(* IEC 61131-3 sources: Industry-PLC-LLM/data/PLCBEAD_repo/PLCBEAD_PLCEmbed-main/PLC-BEAD/Source/GEB/Network_TN_SC_FILL, 1 file *)

(* ---- TN_SC_FILL.ST ---- *)
TYPE
  bya_TN_CHAR:       	ARRAY [0..1919] OF BYTE;
  bya_TN_BACKUP:     	ARRAY [0..1919] OF BYTE;
  bya_TN_COLOR:      	ARRAY [0..1919] OF BYTE;
  bya_TN_Line_Update:	ARRAY [0..23]   OF BOOL;

  us_TN_SCREEN :
  STRUCT
		bya_CHAR:			bya_TN_CHAR;
		bya_COLOR:			bya_TN_COLOR;
		bya_BACKUP:			bya_TN_BACKUP;
		bya_Line_Update:	bya_TN_Line_Update;

		by_Input_Exten_Code:    BYTE;
		by_Input_ASCII_Code:    BYTE;
		bo_Input_ASCII_IsNum:   BOOL;
		in_Page_Number:        	INT;                (* aktive Seiten-Nr.              *)
		in_Cursor_X:           	INT;                (* Cursor X-POSition              *)
		in_Cursor_Y:           	INT;                (* Cursor Y-POSition              *)
		in_EOS_Offset:         	INT;                (* End of String Offset           *)
		by_Clear_Screen_Attr:  	BYTE;               (* Clear-Screen Attr              *)
		bo_Clear_Screen:       	BOOL;               (* Clear-Screen ausl�sen          *)
		bo_Modal_Dialog:       	BOOL;               (* Modaler Dialog ist aktiv       *)
		bo_Menue_Bar_Dialog:   	BOOL;               (* Menue Dialog ist aktiv         *)

  END_STRUCT;
END_TYPE

FUNCTION TN_SC_XY2_ERROR:BOOL

	VAR_INPUT
		X1 :	INT;
		Y1 :	INT;
		X2 :	INT;
		Y2 :	INT;
	END_VAR

	TN_SC_XY2_ERROR := Y1 < 0 OR X1 < 0 OR Y2 < 0 OR X2 < 0 OR Y1 > 23 OR X1 > 79 OR Y2 > 23 OR X2 > 79;

END_FUNCTION

FUNCTION_BLOCK TN_SC_FILL_Block

	VAR
		in_X :	INT;
		in_Y :	INT;
		in_Offset :	INT;
	END_VAR

	VAR_INPUT
		Iin_Y1 :	INT;
		Iin_X1 :	INT;
		Iin_Y2 :	INT;
		Iin_X2 :	INT;
		Iby_CHAR :	BYTE;
		Iby_Attr :	BYTE;
	END_VAR

	VAR_IN_OUT
		Xus_TN_SCREEN :	us_TN_SCREEN;
	END_VAR

	IF TN_SC_XY2_ERROR(Iin_X1,Iin_Y1,Iin_X2,Iin_Y2) THEN RETURN; END_IF;

	FOR in_Y := Iin_Y1 TO Iin_Y2 DO
	Xus_TN_SCREEN.bya_Line_Update[in_Y] := TRUE;
	in_Offset := (in_Y * 80) + Iin_X1;
	FOR in_X := Iin_X1 TO Iin_X2 DO
		Xus_TN_SCREEN.bya_CHAR[in_Offset]  := Iby_CHAR;
		Xus_TN_SCREEN.bya_COLOR[in_Offset] := Iby_Attr;
		in_Offset := in_Offset + 1;
	END_FOR;
	END_FOR;

END_FUNCTION_BLOCK

PROGRAM program0
	VAR
		Iin_Y1 :	INT;
		Iin_X1 :	INT;
		Iin_Y2 :	INT;
		Iin_X2 :	INT;
		Iby_CHAR :	BYTE;
		Iby_Attr :	BYTE;
		Xus_TN_SCREEN :	us_TN_SCREEN;

		func_block : TN_SC_FILL_Block;
	END_VAR
	func_block.Iin_X1 := Iin_X1;
	func_block.Iin_Y1 := Iin_Y1;
  	func_block.Iin_X2 := Iin_X2;
	func_block.Iin_Y2 := Iin_Y2;
  	func_block.Iby_CHAR := Iby_CHAR;
	func_block.Iby_Attr := Iby_Attr;
	func_block.Xus_TN_SCREEN := Xus_TN_SCREEN;

	func_block();
	Xus_TN_SCREEN  := func_block.Xus_TN_SCREEN;
END_PROGRAM
